		3:
		    FilePut_String := '';
			IF (FileWrite_Index = 0) THEN
(*當FileWrite_Index = 0時，代表為文件的第一行。文件的第一行為變數的名稱(Variable_A ~ Variable_I的名稱)*)
				FilePut_String := CONCAT ( Variable_Name[0] , ',' , Variable_Name[1] , ',' , Variable_Name[2] );
				FilePut_String := CONCAT (  FilePut_String , ',' , Variable_Name[3] , ',' , Variable_Name[4] );	
				FilePut_String := CONCAT (  FilePut_String , ',' , Variable_Name[5] , ',' , Variable_Name[6] );	
				FilePut_String := CONCAT (  FilePut_String , ',' , Variable_Name[7] , ',' , Variable_Name[8] );				
			ELSE
(*當FileWrite_Index > 0時，即為Variable_A ~ Variable_I的變數陣列元素儲存*)
			    Variable_A_String := RealToFormatString ( Variable_A[FileWrite_Index-1] , FALSE , TRUE , USINT#2 , USINT#2 );
			    Variable_B_String := RealToFormatString ( Variable_B[FileWrite_Index-1] , FALSE , TRUE , USINT#2 , USINT#2 );
		        Variable_C_String := RealToFormatString ( Variable_C[FileWrite_Index-1] , FALSE , TRUE , USINT#2 , USINT#2 );
			    Variable_D_String := RealToFormatString ( Variable_D[FileWrite_Index-1] , FALSE , TRUE , USINT#2 , USINT#2 );
			    Variable_E_String := RealToFormatString ( Variable_E[FileWrite_Index-1] , FALSE , TRUE , USINT#2 , USINT#2 );
			    Variable_F_String := RealToFormatString ( Variable_F[FileWrite_Index-1] , FALSE , TRUE , USINT#2 , USINT#2 );
			    Variable_G_String :=RealToFormatString ( Variable_G[FileWrite_Index-1] , FALSE , TRUE , USINT#2 , USINT#2 );
			    Variable_H_String :=RealToFormatString ( Variable_H[FileWrite_Index-1] , FALSE , TRUE , USINT#2 , USINT#2 );
			    Variable_I_String := RealToFormatString ( Variable_I[FileWrite_Index-1] , FALSE , TRUE , USINT#2 , USINT#2 );
			
			    FilePut_String := CONCAT (Variable_A_String , ',' , Variable_B_String , ',' , Variable_C_String );
			    FilePut_String :=  CONCAT (  FilePut_String, ',' , Variable_D_String  , ',' , Variable_E_String );
                FilePut_String :=  CONCAT (  FilePut_String, ',' , Variable_F_String  , ',' , Variable_G_String );
			    FilePut_String :=  CONCAT (  FilePut_String, ',' , Variable_H_String  , ',' , Variable_I_String );
			END_IF;
			
			FilePut_String :=  CONCAT (  FilePut_String , '$r$l' );
			  
			 FileWrite_Stage := 4;
		4:
		    FileWrite_Fileput(Execute := TRUE , FileID := FileWrite_FID ,  in := FilePut_String);
			
			IF (  FileWrite_Fileput.Done = TRUE) THEN
			    
				FileWrite_Index :=  FileWrite_Index + 1;
				
				IF (FileWrite_Index <= 10) THEN
					 FileWrite_Fileput(Execute := FALSE );
					 FileWrite_Stage := 3;
				ELSE
					 FileWrite_Stage := 5;
				END_IF;
			END_IF;
			
			IF ( FileWrite_Fileput.Error = TRUE ) THEN
				 FileWrite_Stage :=50;
			END_IF;
		5:
			FileWrite_FileClose(Execute := TRUE , FileID := FileWrite_FID );
			
			IF (FileWrite_FileClose.Done = TRUE ) THEN
				 FileWrite_Busy := FALSE;
			END_IF;
			IF (FileWrite_FileClose.Error = TRUE ) THEN
				 FileWrite_Stage :=50;
			END_IF;			
		50:
		     FileWrite_Busy := FALSE;
	END_CASE;
END_IF;
//*****************************************************************************************
//批次到達時寫入
R_TRIG1(Clk:=Error_BatchOK);
IF R_TRIG1.Q THEN
	nowtime:=_CurrentTime;
	DtToDateStruct(nowtime,nowtimeST);
	File_Name:=CONCAT(UINT_TO_STRING(nowtimeST.Year),UINT_TO_STRING(nowtimeST.Month));
	File_Name:=CONCAT(File_Name,UINT_TO_STRING(nowtimeST.Day));
	File_Name:=CONCAT(File_Name,UINT_TO_STRING(nowtimeST.Hour));
	File_Name:=CONCAT(File_Name,UINT_TO_STRING(nowtimeST.Min));
	File_Name:=CONCAT(File_Name,UINT_TO_STRING(nowtimeST.Sec));
	File_Name_All := CONCAT( File_Name , '.CSV');
	Variable_A[0]:=DINT_TO_REAL(BatchOKCount);
	Variable_B[0]:=DINT_TO_REAL(BatchNGCount);
	Variable_C[0]:=DINT_TO_REAL(BatchTargetCount);
	File_Write_Tri:=TRUE;
END_IF;
IF FileWrite_Busy THEN
	File_Write_Tri:=FALSE;
END_IF;
IF pbsetdt THEN
	sdnt:=dt#2017-12-22-10:56:00.00;
	SetTime(sdnt);
END_IF;
END_PROGRAM

FUNCTION_BLOCK fbErrorDouble
VAR
    TON_1 : TON;
    TON_2 : TON;
END_VAR
VAR_INPUT
    bAutoStatus : BOOL;
    bResetPB : BOOL;
    bBackLS : BOOL;
    bOutLS : BOOL;
    bBackSOL : BOOL;
    bOutSOL : BOOL;
END_VAR
VAR_OUTPUT
    bErrorStatus_Back : BOOL;
    bErrorStatus_Out : BOOL;
END_VAR
IF bAutoStatus AND NOT(bResetPB) THEN
	(*歸磁簧開關*)
	TON_1(IN:=bBackSOL AND NOT(bBackLS), PT:=t#5s);
	IF TON_1.Q THEN
		bErrorStatus_Back:=TRUE;
	END_IF;
	(*出磁簧開關*)
	TON_2(IN:=bOutSOL AND NOT(bOutLS), PT:=t#5s);
	IF TON_2.Q THEN
		bErrorStatus_Out:=TRUE;
	END_IF;
END_IF;
IF bResetPB THEN
	bErrorStatus_Back:=FALSE;
	bErrorStatus_Out:=FALSE;
END_IF;
END_FUNCTION_BLOCK

FUNCTION_BLOCK fbErrorSingle
VAR
    TON_1 : TON;
    TON_2 : TON;
END_VAR
VAR_INPUT
    bAutoStatus : BOOL;
    bResetPB : BOOL;
    bSOL : BOOL;
    bBackLS : BOOL;
    bOutLS : BOOL;
END_VAR
VAR_OUTPUT
    bErrorStatus_Back : BOOL;
    bErrorStatus_Out : BOOL;
END_VAR
IF bAutoStatus AND NOT(bResetPB) THEN
	(*歸磁簧開關*)
	TON_1(IN:=(NOT(bSOL) AND NOT(bBackLS)) OR ((bSOL) AND bBackLS), PT:=t#5s);
	IF TON_1.Q THEN
		bErrorStatus_Back:=TRUE;
	END_IF;
	(*出磁簧開關*)
	TON_2(IN:=(NOT(bSOL) AND (bOutLS)) OR ((bSOL) AND NOT(bOutLS)), PT:=t#5s);
	IF TON_2.Q THEN
		bErrorStatus_Out:=TRUE;
	END_IF;
END_IF;
IF bResetPB THEN
	bErrorStatus_Back:=FALSE;
	bErrorStatus_Out:=FALSE;
END_IF;
END_FUNCTION_BLOCK

FUNCTION_BLOCK fbFull
VAR
    AutoFlow : INT;
    TON_Auto1 : TON;
    TON_Auto2 : TON;
    TON_Auto3 : TON;
    tItemNotExistDelayTime : TIME;
    tItemExistTime : TIME;
    tItemNotExistErrorTime : TIME;
END_VAR
VAR_INPUT
    bFullSNR : BOOL;
    iItemNotExistDelayTime : LINT;
    iItemExistTime : LINT;
    iItemNotExistErrorTime : LINT;
END_VAR
VAR_OUTPUT
    bFullRY : BOOL;
    bFullSNRError : BOOL;
END_VAR
VAR_EXTERNAL
    SystemReadyStatus : BOOL;
END_VAR
(******************************************************************
程式:振動筒程序
作者:蔡相偉
版本資訊:v1.0		2016/4/16
******************************************************************)
//時間轉換
tItemNotExistDelayTime:=NanoSecToTime(In:=iItemNotExistDelayTime*100000000);
tItemExistTime:=NanoSecToTime(In:=iItemExistTime*100000000);
tItemNotExistErrorTime:=NanoSecToTime(In:=iItemNotExistErrorTime*100000000);
(*流程*)
(*PowerOn=0*)
IF NOT(SystemReadyStatus) THEN
	AutoFlow:=0;
END_IF;

(*Idle=1*)
IF AutoFlow=0 AND SystemReadyStatus THEN
	AutoFlow:=1;
END_IF;

IF AutoFlow=3 THEN
	AutoFlow:=1;
END_IF;

(*振動筒起振=2*)
TON_Auto1(IN:=AutoFlow=1 AND NOT(bFullSNR) , PT:=tItemNotExistDelayTime);
IF AutoFlow=1 AND TON_Auto1.Q THEN
	AutoFlow:=2;
END_IF;

(*振動筒停振=3*)
TON_Auto2(IN:=AutoFlow=2 AND bFullSNR , PT:=tItemExistTime);
TON_Auto3(IN:=NOT(bFullSNR) AND bFullRY, PT:=tItemNotExistErrorTime);
IF AutoFlow=2 AND TON_Auto2.Q THEN
	AutoFlow:=3;
END_IF;
(******************************************************************)
(*輸出*)
(*振動筒繼電器*)
IF AutoFlow=2 THEN
	bFullRY:=TRUE;
	ELSE
	bFullRY:=FALSE;
END_IF;
(*振動筒滿料異常*)
IF AutoFlow=2 AND (TON_Auto3.Q) THEN
	bFullSNRError:=TRUE;
	ELSE
	bFullSNRError:=FALSE;
END_IF;
END_FUNCTION_BLOCK

FUNCTION_BLOCK fbFeed
VAR
    tNoObjDelayTime : TIME;
    tObjectExistDelayTime : TIME;
    Autoflow : INT;
    TON_1 : TON;
    TON_2 : TON;
    TON_3 : TON;
    ObjSNRStatus : BOOL;
    THStatus : BOOL;
    R_TRIG_1 : R_TRIG;
    R_TRIG_2 : R_TRIG;
    R_TRIG_3 : R_TRIG;
    R_TRIG_4 : R_TRIG;
END_VAR
VAR_INPUT
    wNoObjDelayTime : LINT;
    wObjectExistDelayTime : LINT;
    bReset : BOOL;
    bTHPB : BOOL;
    bObjSNR : BOOL;
    bFeedStart : BOOL;
    bTHBackLS : BOOL;
    bTHOutLS : BOOL;
    bErrorTHBack : BOOL;
    bErrorTHOut : BOOL;
    bInterlock_thback : BOOL;
    bInterlock_thout : BOOL;
    bSupplierRY : BOOL;
END_VAR
VAR_OUTPUT
    bFeedError : BOOL;
    bFeedFinish : BOOL;
    bTHSOL : BOOL;
    bFeedRY : BOOL;
END_VAR
VAR_EXTERNAL
    SystemReadyStatus : BOOL;
    AutoStatus : BOOL;
END_VAR
(*************************************************************************
程序名稱:平送FB
作者:蔡相偉
版本,日期,版本資訊:
1.0.0	2016/6/28		初始版本

PowerOn=0
Idle=1
無料,節流出=2
到出,平送起振=3
工件到位,平送停振=4
節流回=5
節流到回=6
*************************************************************************)
//時間轉換
tNoObjDelayTime:=NanoSecToTime(wNoObjDelayTime*100000000);
tObjectExistDelayTime:=NanoSecToTime(wObjectExistDelayTime*100000000);

//PowerOn=0
IF Autoflow=0 AND SystemReadyStatus AND NOT(bErrorTHBack) AND NOT(bErrorTHOut) AND AutoStatus  THEN
	Autoflow:=1;
END_IF;

(*Idle=1*)
TON_1(IN:= Autoflow=1 AND NOT(bObjSNR) ,PT:= tNoObjDelayTime);
IF Autoflow=1 AND (bFeedStart) THEN
	Autoflow:=2;
END_IF;
(*無料,節流出=2*)
IF Autoflow=2 THEN
	ObjSNRStatus:=FALSE;
END_IF;

IF Autoflow=2 AND bTHOutLS THEN
	Autoflow:=3;
END_IF;
(*到出,平送起振=3*)
IF Autoflow=3 AND bObjSNR THEN
	ObjSNRStatus:=TRUE;
END_IF;
TON_2(IN:= Autoflow=3 AND bObjSNR ,PT:= tObjectExistDelayTime);
TON_3(IN:= Autoflow=3 AND NOT(bObjSNR) ,PT:= t#4s);
IF TON_3.Q THEN
	bFeedError:=TRUE;
END_IF;
IF bReset THEN
	bFeedError:=FALSE;
END_IF;

IF Autoflow=3 AND TON_2.Q AND NOT(bFeedError) THEN
	Autoflow:=4;
END_IF;
(*工件到位,平送停振=4*)
IF Autoflow=4 THEN
	Autoflow:=5;
END_IF;
(*節流回=5*)
IF Autoflow=5 AND bTHBackLS THEN
	Autoflow:=6;
END_IF;
(*節流到回=6*)
IF Autoflow=6 THEN
	bFeedFinish:=TRUE;
	ELSE
	bFeedFinish:=FALSE;
END_IF;

IF Autoflow=6 AND NOT(bFeedStart) THEN
	Autoflow:=1;
END_IF;
(*************************************************************************)
(*Error*)
R_TRIG_3(CLK:=bErrorTHBack);
R_TRIG_4(CLK:=bErrorTHOut);

IF NOT(SystemReadyStatus) OR NOT(AutoStatus) OR bErrorTHBack OR bErrorTHOut THEN
	Autoflow:=0;
END_IF;

(*************************************************************************)
(*手動*)
(*節流*)
R_TRIG_1(CLK:=bTHPB AND NOT(AutoStatus));
(*SET*)
IF (((R_TRIG_1.Q) AND NOT(THStatus)) OR Autoflow=2 OR R_TRIG_3.Q) AND bInterlock_thout THEN
	bTHSOL:=TRUE;
END_IF;
(*RESET*)
IF (((R_TRIG_1.Q) AND THStatus) OR Autoflow=5 OR R_TRIG_4.Q) AND bInterlock_thback THEN
	bTHSOL:=FALSE;
END_IF;
(*STATE*)
THStatus:=bTHSOL;

(*平送*)
(*輸出*)
bFeedRY:=Autoflow=2 OR Autoflow=3 OR bSupplierRY OR bTHSOL;
END_FUNCTION_BLOCK